FUNCTION_BLOCK FB_HomePrepare
VAR_INPUT
    En: BOOL;
    bReset: BOOL;
    bExecute: BOOL;
    nCmdData: UINT;
END_VAR
VAR_IN_OUT
    Axis: AXIS_REF;
END_VAR
VAR_OUTPUT
    EnO: BOOL;
    bBusy: BOOL;
    bDone: BOOL;
    bError: BOOL;
    nErrorId: UDINT;
    bSofLimEnableLowOriginal: BOOL:=TRUE;
    bSofLimEnableHighOriginal: BOOL:=TRUE;
    fVelocityToCam: LREAL:=0;
    fVelocityFromCam: LREAL:=0;
END_VAR
VAR
    fbHomeReadSoftLimEnable:FB_HomeReadSoftLimEnable;
    fbHomeDisableSoftLimEnable:FB_HomeWriteSoftLimEnable;
    fbHomeReadNCVelocities: FB_HomeReadNcVelocities;
    fbHomeResetCalibrationFlag:MC_Home;   //Only used for reset of calibration flag
    fbExecuteRiseEdge: R_TRIG;
    bExecuteReadNC:BOOL:=FALSE;
    bExecuteWriteNC:BOOL:=FALSE;
    nState:INT:=0;
END_VAR

En:=EnO;
IF bReset THEN
    bError:=FALSE;
    nErrorId:=0;
END_IF

IF NOT bExecute THEN
  bExecuteReadNC:=FALSE;
  bExecuteWriteNC:=FALSE;
  nState:=0;
END_IF

fbExecuteRiseEdge(CLK:=bExecute);
IF fbExecuteRiseEdge.Q THEN
  bExecuteReadNC:=TRUE;
END_IF

// Read from NC
fbHomeReadNCVelocities(
  En:=En,
  bExecute:=bExecuteReadNC, // Actualy not needed for sequence 15 (set position only, no movement))
  bReset:=bReset,
  Axis:=Axis,
);

fbHomeReadSoftLimEnable(
    En:=En,
    bExecute:=bExecuteReadNC AND bExecute,
    Axis:=Axis,
    bReset:=bReset,
);

// Reset calibration flag
fbHomeResetCalibrationFlag(
  Execute:=bExecuteReadNC,
  HomingMode:=MC_ResetCalibration,
  Axis:=Axis
);

bSofLimEnableLowOriginal:=fbHomeReadSoftLimEnable.bSofLimEnableLow;
bSofLimEnableHighOriginal:=fbHomeReadSoftLimEnable.bSofLimEnableHigh;

fVelocityToCam:=fbHomeReadNCVelocities.fVelocityToCam;
fVelocityFromCam:=fbHomeReadNCVelocities.fVelocityFromCam;

IF bExecuteReadNC AND bExecute AND fbHomeReadSoftLimEnable.bDone THEN
    fbHomeDisableSoftLimEnable.bSofLimEnableHigh:=FALSE;
    fbHomeDisableSoftLimEnable.bSofLimEnableLow:=FALSE;
    bExecuteWriteNC:=TRUE; //Always write (only needed if enabled actually)
END_IF

// Write to NC (disable soft limits)
fbHomeDisableSoftLimEnable(
    En:=En,
    bExecute:=bExecuteWriteNC AND bExecute,
    Axis:=Axis,
    bReset:=bReset,
);

bBusy:=fbHomeReadSoftLimEnable.bBusy OR fbHomeDisableSoftLimEnable.bBusy OR fbHomeReadNCVelocities.bBusy OR fbHomeResetCalibrationFlag.Busy;
bDone:=fbHomeReadSoftLimEnable.bDone AND fbHomeDisableSoftLimEnable.bDone AND fbHomeReadNCVelocities.bDone AND fbHomeResetCalibrationFlag.Done AND bExecute;

bError:=fbHomeReadSoftLimEnable.bError OR fbHomeDisableSoftLimEnable.bError OR fbHomeReadNCVelocities.bError OR fbHomeResetCalibrationFlag.Error;
IF fbHomeReadSoftLimEnable.bError THEN
  nErrorId:=fbHomeReadSoftLimEnable.nErrorId;
ELSIF fbHomeDisableSoftLimEnable.bError THEN
  nErrorId:=fbHomeDisableSoftLimEnable.nErrorId;
ELSIF fbHomeResetCalibrationFlag.Error THEN
  nErrorId:=fbHomeResetCalibrationFlag.ErrorId;
END_IF

END_FUNCTION_BLOCK

(* stored: Version 1.1.0.1, ProductVersion 3.1.4024.0
   POU FB_HomePrepare: Id {44b4f5e1-854c-4705-82a0-c1e3db13fb33}, SpecialFunc None *)
